TYPE SafetyStatuses :
STRUCT
	initializationStatus: InitializationStatus;
	healthStatus: HealthStatus;
	busyStatus: BusyStatus;
	operatingStatus: OperatingStatus;
	communicationHealthStatus: HealthStatus;
	functionBlockHealthStatus: HealthStatus;
	outputHealthStatus: HealthStatus;
END_STRUCT
END_TYPE

(* stored: Version 1.1.0.1, ProductVersion 3.1.4019.2
   DUT SafetyStatuses: Id {17126cfb-82c8-4e79-9809-e1bb43eb71ea} *)
